// Mitsubishi GX Works2 project: PROGRAM COBA COBA COBA HMI aja   PLC: FX3U/FX3UC

PROGRAM MAIN
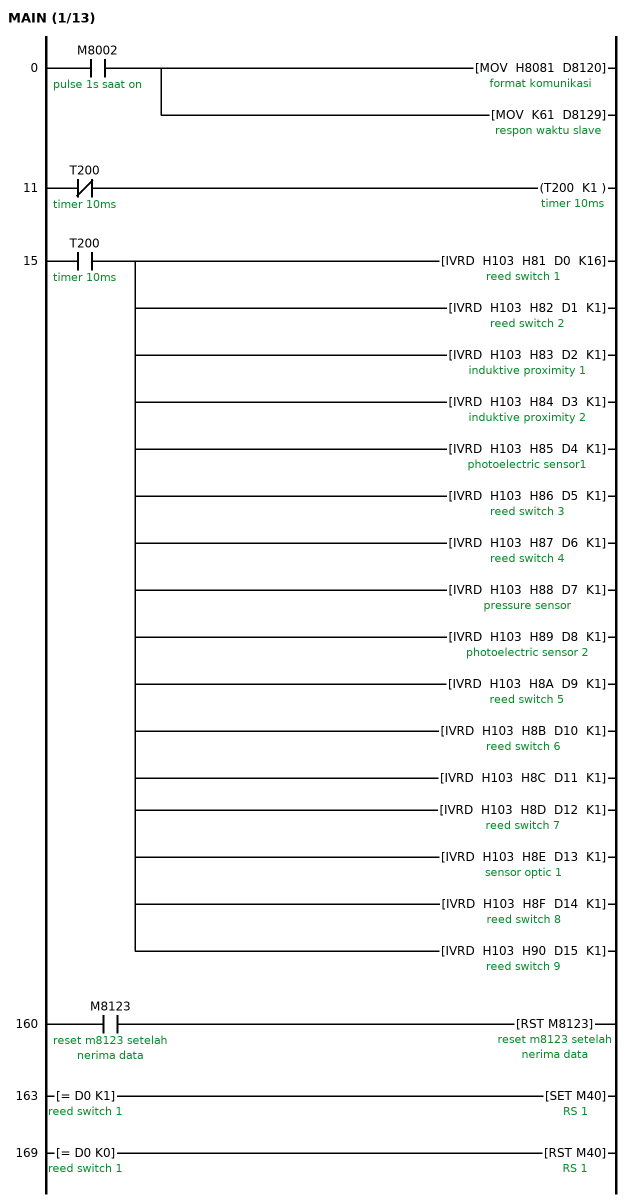
0     LD      M8002  ; pulse 1s saat on
      MOV     H8081 D8120  ; format komunikasi
      MOV     K61 D8129  ; respon waktu slave
11    LDI     T200  ; timer 10ms
      OUT     T200 K1  ; timer 10ms
15    LD      T200  ; timer 10ms
      IVRD    H103 H81 D0 K16  ; reed switch 1
      IVRD    H103 H82 D1 K1  ; reed switch 2
      IVRD    H103 H83 D2 K1  ; induktive proximity 1
      IVRD    H103 H84 D3 K1  ; induktive proximity 2
      IVRD    H103 H85 D4 K1  ; photoelectric sensor1
      IVRD    H103 H86 D5 K1  ; reed switch 3
      IVRD    H103 H87 D6 K1  ; reed switch 4
      IVRD    H103 H88 D7 K1  ; pressure sensor
      IVRD    H103 H89 D8 K1  ; photoelectric sensor 2
      IVRD    H103 H8A D9 K1  ; reed switch 5
      IVRD    H103 H8B D10 K1  ; reed switch 6
      IVRD    H103 H8C D11 K1
      IVRD    H103 H8D D12 K1  ; reed switch 7
      IVRD    H103 H8E D13 K1  ; sensor optic 1
      IVRD    H103 H8F D14 K1  ; reed switch 8
      IVRD    H103 H90 D15 K1  ; reed switch 9
160   LD      M8123  ; reset m8123 setelah nerima data
      RST     M8123  ; reset m8123 setelah nerima data
163   LD=     D0 K1  ; reed switch 1
      SET     M40  ; RS 1
169   LD=     D0 K0  ; reed switch 1
      RST     M40  ; RS 1
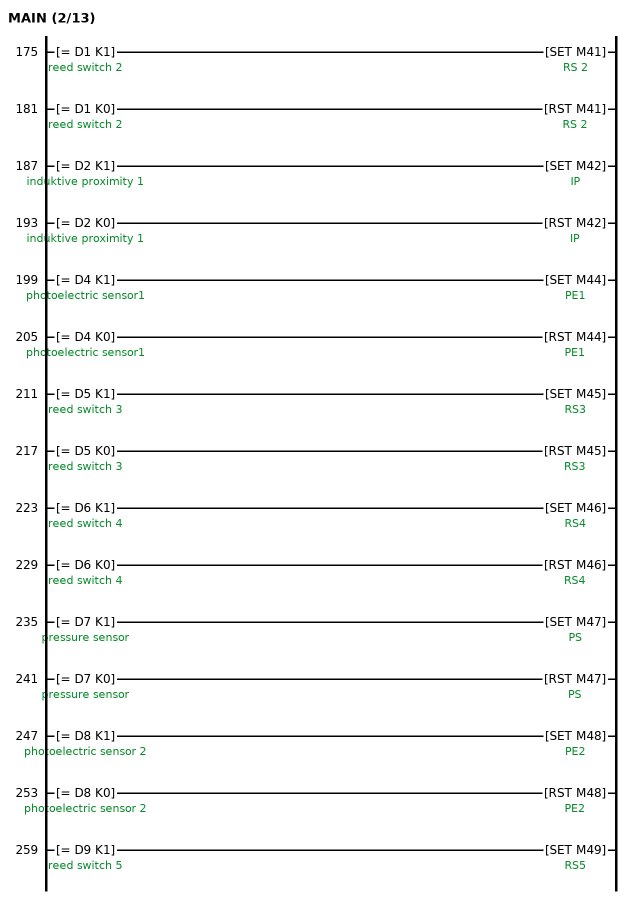
175   LD=     D1 K1  ; reed switch 2
      SET     M41  ; RS 2
181   LD=     D1 K0  ; reed switch 2
      RST     M41  ; RS 2
187   LD=     D2 K1  ; induktive proximity 1
      SET     M42  ; IP
193   LD=     D2 K0  ; induktive proximity 1
      RST     M42  ; IP
199   LD=     D4 K1  ; photoelectric sensor1
      SET     M44  ; PE1
205   LD=     D4 K0  ; photoelectric sensor1
      RST     M44  ; PE1
211   LD=     D5 K1  ; reed switch 3
      SET     M45  ; RS3
217   LD=     D5 K0  ; reed switch 3
      RST     M45  ; RS3
223   LD=     D6 K1  ; reed switch 4
      SET     M46  ; RS4
229   LD=     D6 K0  ; reed switch 4
      RST     M46  ; RS4
235   LD=     D7 K1  ; pressure sensor
      SET     M47  ; PS
241   LD=     D7 K0  ; pressure sensor
      RST     M47  ; PS
247   LD=     D8 K1  ; photoelectric sensor 2
      SET     M48  ; PE2
253   LD=     D8 K0  ; photoelectric sensor 2
      RST     M48  ; PE2
259   LD=     D9 K1  ; reed switch 5
      SET     M49  ; RS5
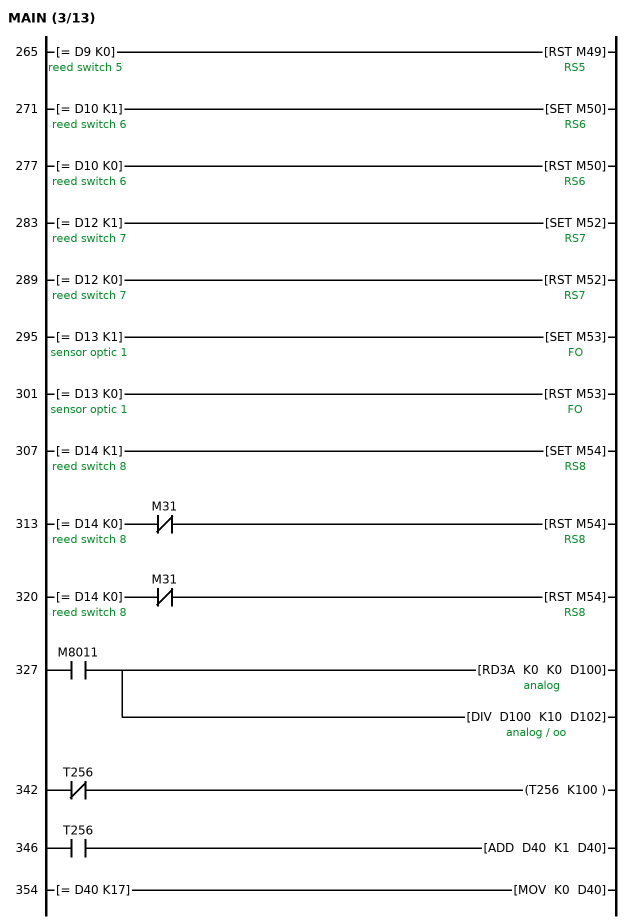
265   LD=     D9 K0  ; reed switch 5
      RST     M49  ; RS5
271   LD=     D10 K1  ; reed switch 6
      SET     M50  ; RS6
277   LD=     D10 K0  ; reed switch 6
      RST     M50  ; RS6
283   LD=     D12 K1  ; reed switch 7
      SET     M52  ; RS7
289   LD=     D12 K0  ; reed switch 7
      RST     M52  ; RS7
295   LD=     D13 K1  ; sensor optic 1
      SET     M53  ; FO
301   LD=     D13 K0  ; sensor optic 1
      RST     M53  ; FO
307   LD=     D14 K1  ; reed switch 8
      SET     M54  ; RS8
313   LD=     D14 K0  ; reed switch 8
      ANI     M31
      RST     M54  ; RS8
320   LD=     D14 K0  ; reed switch 8
      ANI     M31
      RST     M54  ; RS8
327   LD      M8011
      RD3A    K0 K0 D100  ; analog
      DIV     D100 K10 D102  ; oo
342   LDI     T256
      OUT     T256 K100
346   LD      T256
      ADD     D40 K1 D40
354   LD=     D40 K17
      MOV     K0 D40
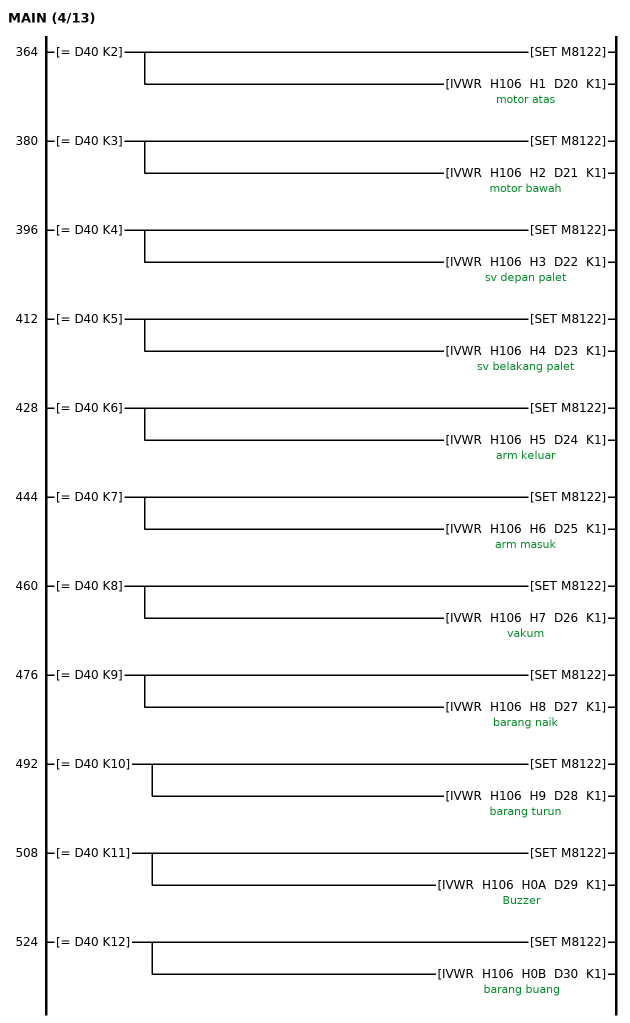
364   LD=     D40 K2
      SET     M8122
      IVWR    H106 H1 D20 K1  ; motor atas
380   LD=     D40 K3
      SET     M8122
      IVWR    H106 H2 D21 K1  ; motor bawah
396   LD=     D40 K4
      SET     M8122
      IVWR    H106 H3 D22 K1  ; sv depan palet
412   LD=     D40 K5
      SET     M8122
      IVWR    H106 H4 D23 K1  ; sv belakang palet
428   LD=     D40 K6
      SET     M8122
      IVWR    H106 H5 D24 K1  ; arm keluar
444   LD=     D40 K7
      SET     M8122
      IVWR    H106 H6 D25 K1  ; arm masuk
460   LD=     D40 K8
      SET     M8122
      IVWR    H106 H7 D26 K1  ; vakum
476   LD=     D40 K9
      SET     M8122
      IVWR    H106 H8 D27 K1  ; barang naik
492   LD=     D40 K10
      SET     M8122
      IVWR    H106 H9 D28 K1  ; barang turun
508   LD=     D40 K11
      SET     M8122
      IVWR    H106 H0A D29 K1  ; Buzzer
524   LD=     D40 K12
      SET     M8122
      IVWR    H106 H0B D30 K1  ; barang buang
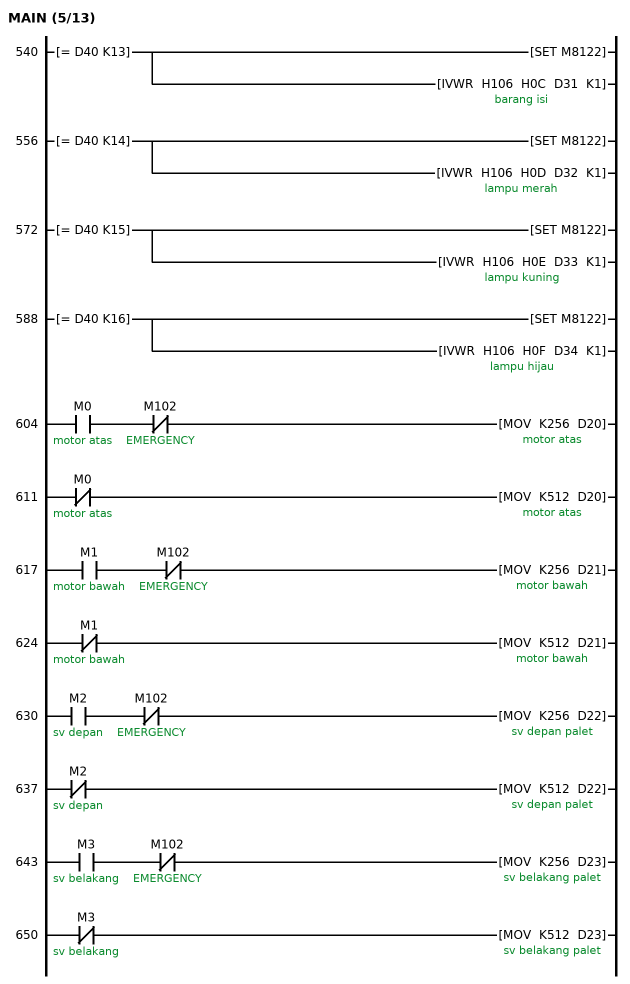
540   LD=     D40 K13
      SET     M8122
      IVWR    H106 H0C D31 K1  ; barang isi
556   LD=     D40 K14
      SET     M8122
      IVWR    H106 H0D D32 K1  ; lampu merah
572   LD=     D40 K15
      SET     M8122
      IVWR    H106 H0E D33 K1  ; lampu kuning
588   LD=     D40 K16
      SET     M8122
      IVWR    H106 H0F D34 K1  ; lampu hijau
604   LD      M0  ; motor atas
      ANI     M102  ; EMERGENCY
      MOV     K256 D20
611   LDI     M0  ; motor atas
      MOV     K512 D20
617   LD      M1  ; motor bawah
      ANI     M102  ; EMERGENCY
      MOV     K256 D21
624   LDI     M1  ; motor bawah
      MOV     K512 D21
630   LD      M2  ; sv depan
      ANI     M102  ; EMERGENCY
      MOV     K256 D22
637   LDI     M2  ; sv depan
      MOV     K512 D22
643   LD      M3  ; sv belakang
      ANI     M102  ; EMERGENCY
      MOV     K256 D23
650   LDI     M3  ; sv belakang
      MOV     K512 D23
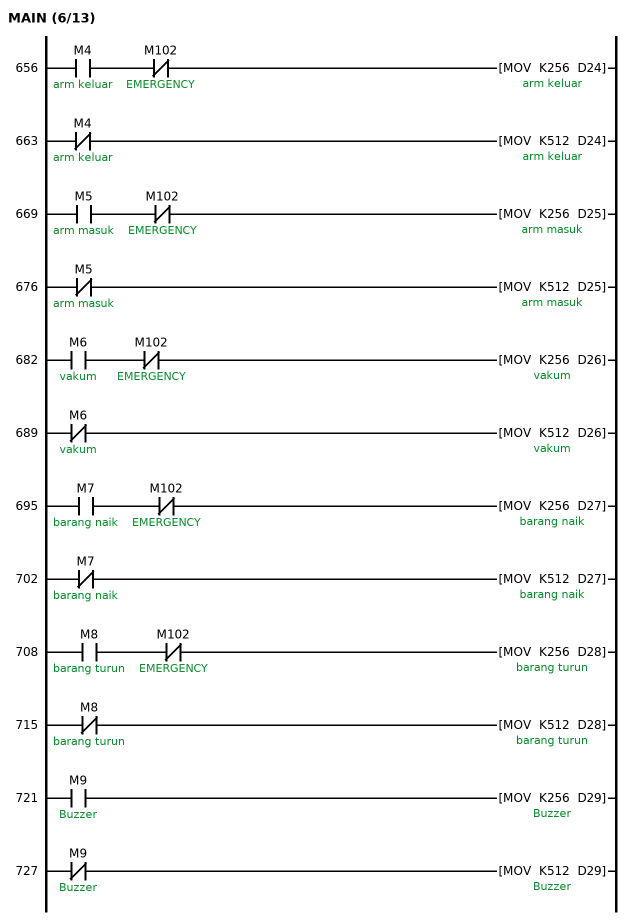
656   LD      M4  ; arm keluar
      ANI     M102  ; EMERGENCY
      MOV     K256 D24
663   LDI     M4  ; arm keluar
      MOV     K512 D24
669   LD      M5  ; arm masuk
      ANI     M102  ; EMERGENCY
      MOV     K256 D25
676   LDI     M5  ; arm masuk
      MOV     K512 D25
682   LD      M6  ; vakum
      ANI     M102  ; EMERGENCY
      MOV     K256 D26
689   LDI     M6  ; vakum
      MOV     K512 D26
695   LD      M7  ; barang naik
      ANI     M102  ; EMERGENCY
      MOV     K256 D27
702   LDI     M7  ; barang naik
      MOV     K512 D27
708   LD      M8  ; barang turun
      ANI     M102  ; EMERGENCY
      MOV     K256 D28
715   LDI     M8  ; barang turun
      MOV     K512 D28
721   LD      M9  ; Buzzer
      MOV     K256 D29
727   LDI     M9  ; Buzzer
      MOV     K512 D29
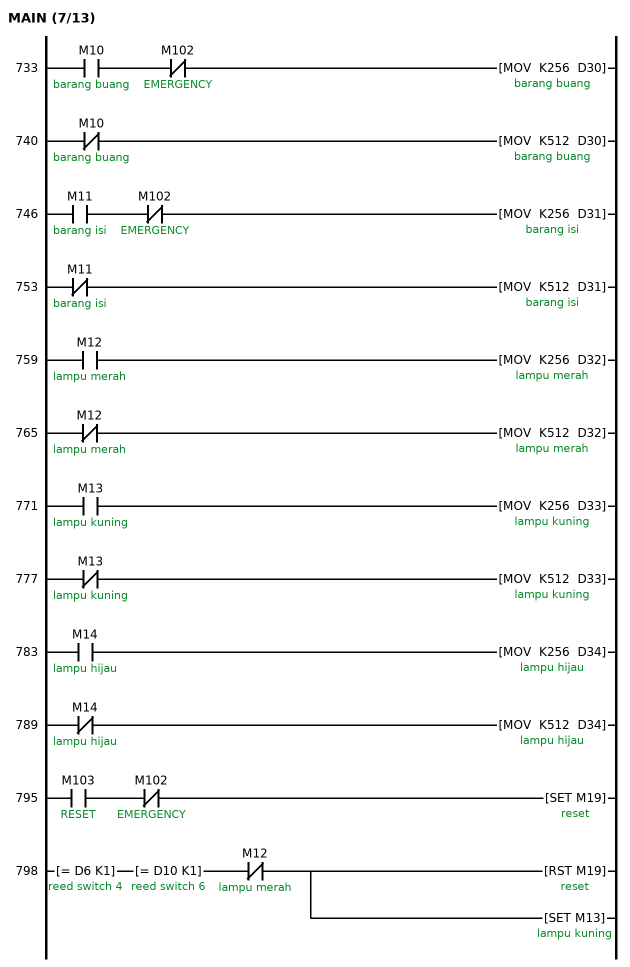
733   LD      M10  ; barang buang
      ANI     M102  ; EMERGENCY
      MOV     K256 D30
740   LDI     M10  ; barang buang
      MOV     K512 D30
746   LD      M11  ; barang isi
      ANI     M102  ; EMERGENCY
      MOV     K256 D31
753   LDI     M11  ; barang isi
      MOV     K512 D31
759   LD      M12  ; lampu merah
      MOV     K256 D32
765   LDI     M12  ; lampu merah
      MOV     K512 D32
771   LD      M13  ; lampu kuning
      MOV     K256 D33
777   LDI     M13  ; lampu kuning
      MOV     K512 D33
783   LD      M14  ; lampu hijau
      MOV     K256 D34
789   LDI     M14  ; lampu hijau
      MOV     K512 D34
795   LD      M103  ; RESET
      ANI     M102  ; EMERGENCY
      SET     M19  ; reset
798   LD=     D6 K1  ; reed switch 4
      AND=    D10 K1  ; reed switch 6
      ANI     M12  ; lampu merah
      RST     M19  ; reset
      SET     M13  ; lampu kuning
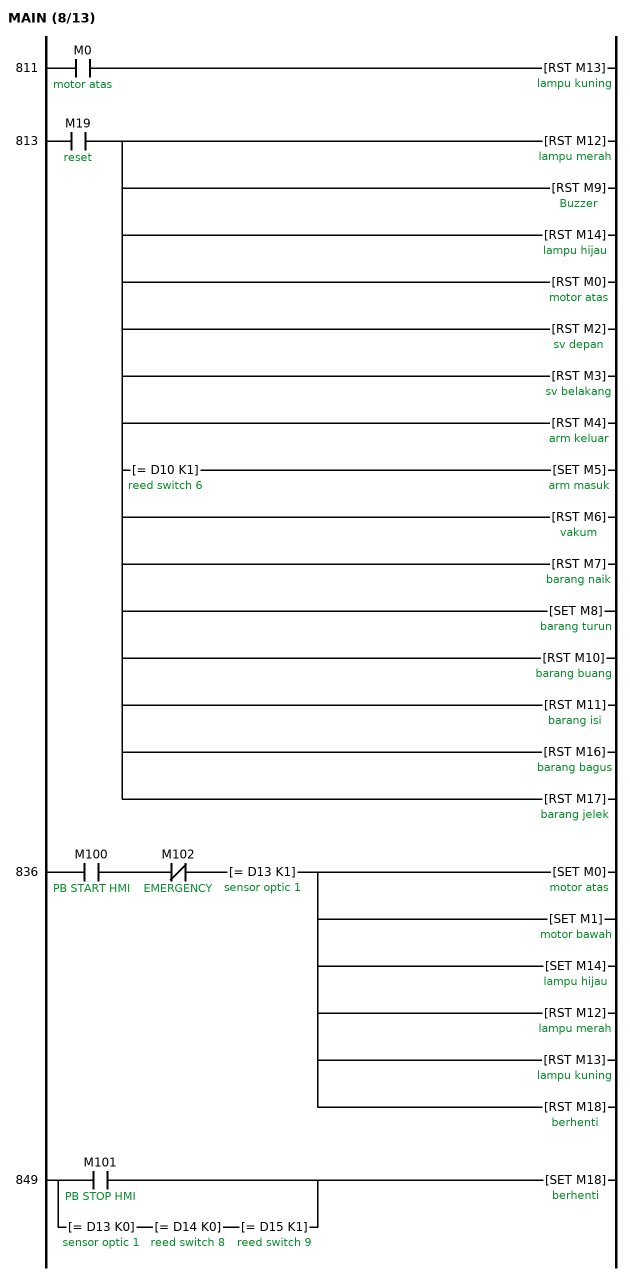
811   LD      M0  ; motor atas
      RST     M13  ; lampu kuning
813   LD      M19  ; reset
      RST     M12  ; lampu merah
      RST     M9  ; Buzzer
      RST     M14  ; lampu hijau
      RST     M0  ; motor atas
      RST     M2  ; sv depan
      RST     M3  ; sv belakang
      RST     M4  ; arm keluar
      MPS
      AND=    D10 K1  ; reed switch 6
      SET     M5  ; arm masuk
      MPP
      RST     M6  ; vakum
      RST     M7  ; barang naik
      SET     M8  ; barang turun
      RST     M10  ; barang buang
      RST     M11  ; barang isi
      RST     M16  ; barang bagus
      RST     M17  ; barang jelek
836   LD      M100  ; PB START HMI
      ANI     M102  ; EMERGENCY
      AND=    D13 K1  ; sensor optic 1
      SET     M0  ; motor atas
      SET     M1  ; motor bawah
      SET     M14  ; lampu hijau
      RST     M12  ; lampu merah
      RST     M13  ; lampu kuning
      RST     M18  ; berhenti
849   LD      M101  ; PB STOP HMI
      LD=     D13 K0  ; sensor optic 1
      AND=    D14 K0  ; reed switch 8
      AND=    D15 K1  ; reed switch 9
      ORB
      SET     M18  ; berhenti
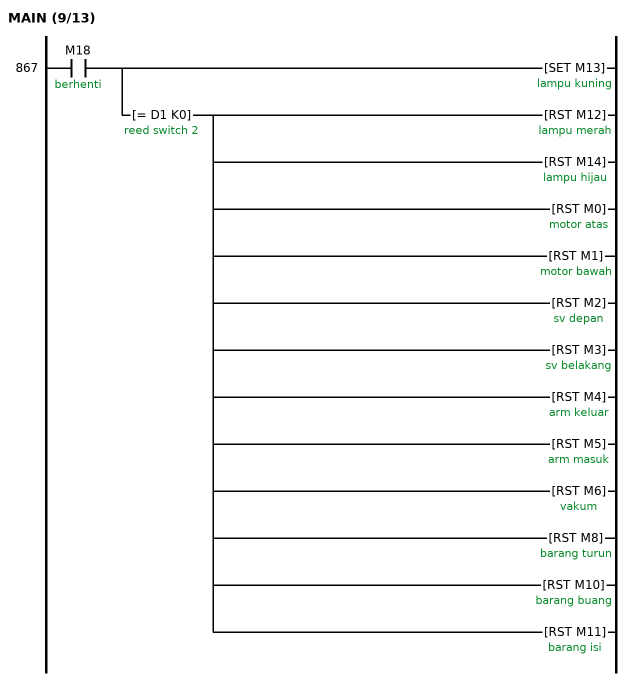
867   LD      M18  ; berhenti
      SET     M13  ; lampu kuning
      AND=    D1 K0  ; reed switch 2
      RST     M12  ; lampu merah
      RST     M14  ; lampu hijau
      RST     M0  ; motor atas
      RST     M1  ; motor bawah
      RST     M2  ; sv depan
      RST     M3  ; sv belakang
      RST     M4  ; arm keluar
      RST     M5  ; arm masuk
      RST     M6  ; vakum
      RST     M8  ; barang turun
      RST     M10  ; barang buang
      RST     M11  ; barang isi
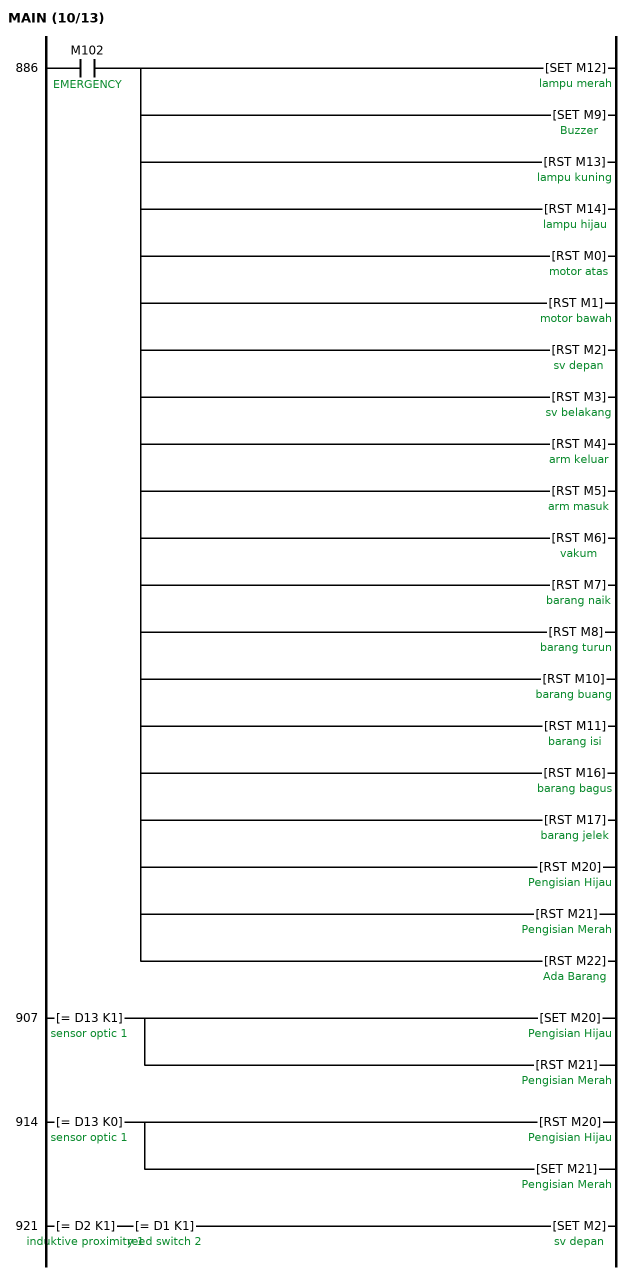
886   LD      M102  ; EMERGENCY
      SET     M12  ; lampu merah
      SET     M9  ; Buzzer
      RST     M13  ; lampu kuning
      RST     M14  ; lampu hijau
      RST     M0  ; motor atas
      RST     M1  ; motor bawah
      RST     M2  ; sv depan
      RST     M3  ; sv belakang
      RST     M4  ; arm keluar
      RST     M5  ; arm masuk
      RST     M6  ; vakum
      RST     M7  ; barang naik
      RST     M8  ; barang turun
      RST     M10  ; barang buang
      RST     M11  ; barang isi
      RST     M16  ; barang bagus
      RST     M17  ; barang jelek
      RST     M20  ; Pengisian Hijau
      RST     M21  ; Pengisian Merah
      RST     M22  ; Ada Barang
907   LD=     D13 K1  ; sensor optic 1
      SET     M20  ; Pengisian Hijau
      RST     M21  ; Pengisian Merah
914   LD=     D13 K0  ; sensor optic 1
      RST     M20  ; Pengisian Hijau
      SET     M21  ; Pengisian Merah
921   LD=     D2 K1  ; induktive proximity 1
      AND=    D1 K1  ; reed switch 2
      SET     M2  ; sv depan
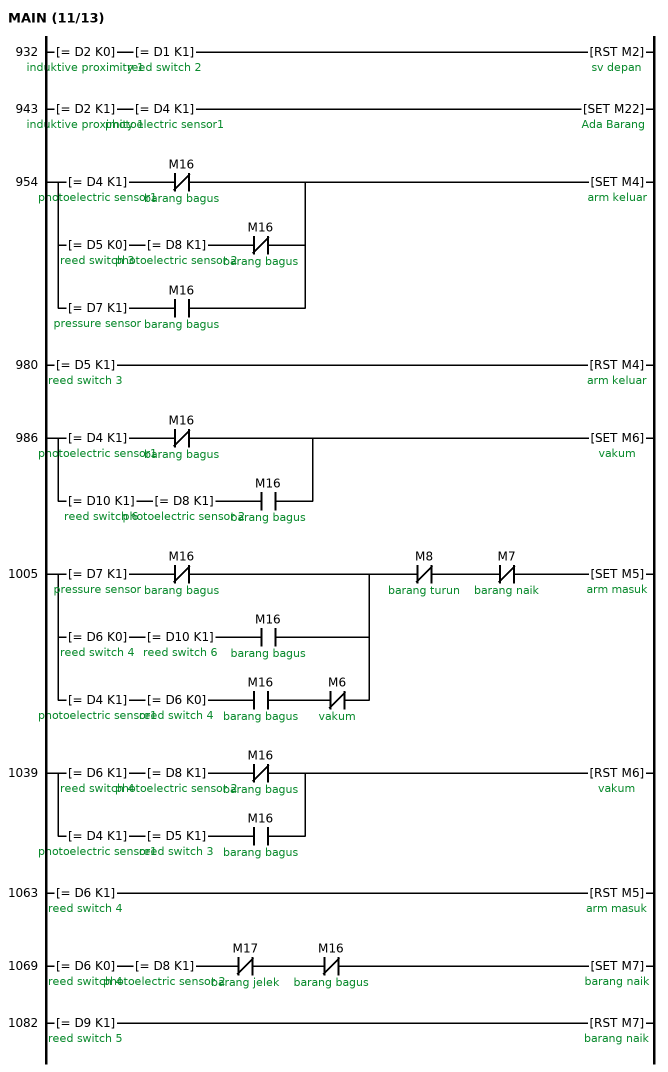
932   LD=     D2 K0  ; induktive proximity 1
      AND=    D1 K1  ; reed switch 2
      RST     M2  ; sv depan
943   LD=     D2 K1  ; induktive proximity 1
      AND=    D4 K1  ; photoelectric sensor1
      SET     M22  ; Ada Barang
954   LD=     D4 K1  ; photoelectric sensor1
      ANI     M16  ; barang bagus
      LD=     D5 K0  ; reed switch 3
      AND=    D8 K1  ; photoelectric sensor 2
      ANI     M16  ; barang bagus
      ORB
      LD=     D7 K1  ; pressure sensor
      AND     M16  ; barang bagus
      ORB
      SET     M4  ; arm keluar
980   LD=     D5 K1  ; reed switch 3
      RST     M4  ; arm keluar
986   LD=     D4 K1  ; photoelectric sensor1
      ANI     M16  ; barang bagus
      LD=     D10 K1  ; reed switch 6
      AND=    D8 K1  ; photoelectric sensor 2
      AND     M16  ; barang bagus
      ORB
      SET     M6  ; vakum
1005  LD=     D7 K1  ; pressure sensor
      ANI     M16  ; barang bagus
      LD=     D6 K0  ; reed switch 4
      AND=    D10 K1  ; reed switch 6
      AND     M16  ; barang bagus
      ORB
      LD=     D4 K1  ; photoelectric sensor1
      AND=    D6 K0  ; reed switch 4
      AND     M16  ; barang bagus
      ANI     M6  ; vakum
      ORB
      ANI     M8  ; barang turun
      ANI     M7  ; barang naik
      SET     M5  ; arm masuk
1039  LD=     D6 K1  ; reed switch 4
      AND=    D8 K1  ; photoelectric sensor 2
      ANI     M16  ; barang bagus
      LD=     D4 K1  ; photoelectric sensor1
      AND=    D5 K1  ; reed switch 3
      AND     M16  ; barang bagus
      ORB
      RST     M6  ; vakum
1063  LD=     D6 K1  ; reed switch 4
      RST     M5  ; arm masuk
1069  LD=     D6 K0  ; reed switch 4
      AND=    D8 K1  ; photoelectric sensor 2
      ANI     M17  ; barang jelek
      ANI     M16  ; barang bagus
      SET     M7  ; barang naik
1082  LD=     D9 K1  ; reed switch 5
      RST     M7  ; barang naik
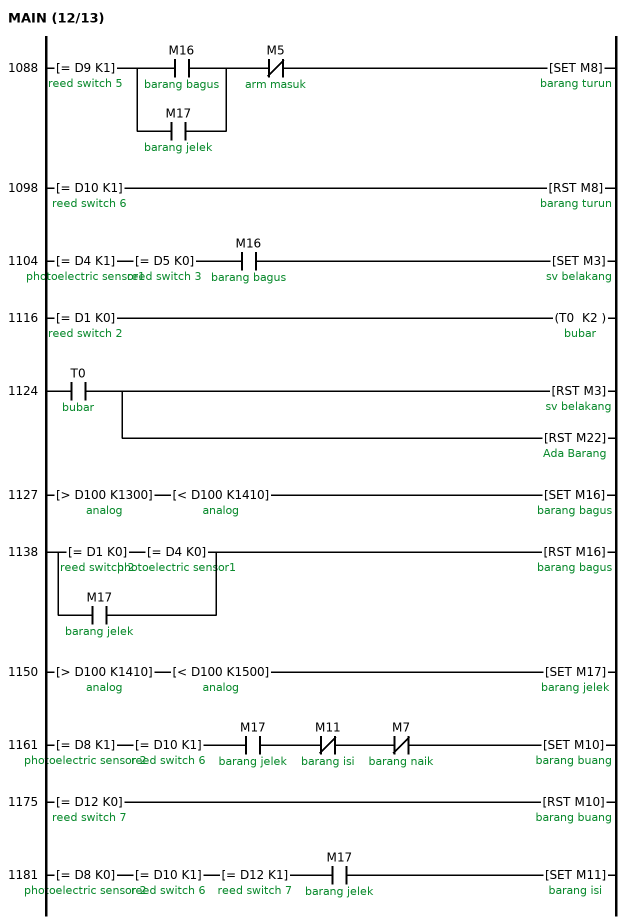
1088  LD=     D9 K1  ; reed switch 5
      LD      M16  ; barang bagus
      OR      M17  ; barang jelek
      ANB
      ANI     M5  ; arm masuk
      SET     M8  ; barang turun
1098  LD=     D10 K1  ; reed switch 6
      RST     M8  ; barang turun
1104  LD=     D4 K1  ; photoelectric sensor1
      AND=    D5 K0  ; reed switch 3
      AND     M16  ; barang bagus
      SET     M3  ; sv belakang
1116  LD=     D1 K0  ; reed switch 2
      OUT     T0 K2  ; bubar
1124  LD      T0  ; bubar
      RST     M3  ; sv belakang
      RST     M22  ; Ada Barang
1127  LD>     D100 K1300  ; analog
      AND<    D100 K1410  ; analog
      SET     M16  ; barang bagus
1138  LD=     D1 K0  ; reed switch 2
      AND=    D4 K0  ; photoelectric sensor1
      OR      M17  ; barang jelek
      RST     M16  ; barang bagus
1150  LD>     D100 K1410  ; analog
      AND<    D100 K1500  ; analog
      SET     M17  ; barang jelek
1161  LD=     D8 K1  ; photoelectric sensor 2
      AND=    D10 K1  ; reed switch 6
      AND     M17  ; barang jelek
      ANI     M11  ; barang isi
      ANI     M7  ; barang naik
      SET     M10  ; barang buang
1175  LD=     D12 K0  ; reed switch 7
      RST     M10  ; barang buang
1181  LD=     D8 K0  ; photoelectric sensor 2
      AND=    D10 K1  ; reed switch 6
      AND=    D12 K1  ; reed switch 7
      AND     M17  ; barang jelek
      SET     M11  ; barang isi
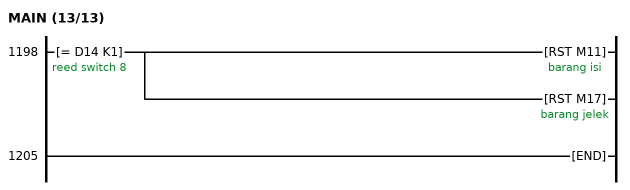
1198  LD=     D14 K1  ; reed switch 8
      RST     M11  ; barang isi
      RST     M17  ; barang jelek
1205  END
END_PROGRAM

// device comments not shown above
X000  ; PB START
X001  ; PB STOP
X002  ; PB RESET
X003  ; emergency
M43  ; IP2
M55  ; RS9
D16  ; motor
D17  ; sv belakang
T220  ; delay arm masuk
C0  ; counter barang
